{region '#Template'}
	{attribute 'Version' := '5.1.0.0'}
	{attribute 'Tags' := '"LCID": "1031", "Text": "Gebäudeautomation, Kommunikation, Server, Client, Publisher, Subscriber"'}
	{attribute 'Tags' := '"LCID": "1033", "Text": "Building automation, Communication, Server, Client, Publisher, Subscriber"'}
	{attribute 'Using' := '"Type": "Template", "URI": "Site"'}
	{attribute 'Description' := '"LCID": "1031", "Text": "Server Datenkommunikation"'}
	{attribute 'Description' := '"LCID": "1033", "Text": "Server data communication"'}
{endregion}

FUNCTION_BLOCK FB_BA_AdsComServer_Room
VAR_INPUT CONSTANT
  	BuildingEnergyLevel		: FB_BA_RawPublisher;
	BuildingSpRmT			: FB_BA_RawPublisher;
	BuildingLighting		: FB_BA_RawPublisher;
END_VAR

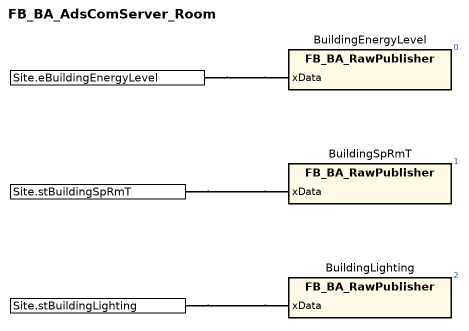
BuildingEnergyLevel(xData := Site.eBuildingEnergyLevel); // FB_BA_RawPublisher
BuildingSpRmT(xData := Site.stBuildingSpRmT); // FB_BA_RawPublisher
BuildingLighting(xData := Site.stBuildingLighting); // FB_BA_RawPublisher

END_FUNCTION_BLOCK

(* stored: Version 1.1.0.1, ProductVersion 3.1.4024.12
   POU FB_BA_AdsComServer_Room: Id {dfa5c561-43c6-4aa0-b664-dc4628b7cadf}, SpecialFunc None *)
